// TIA Portal V17 export
FUNCTION_BLOCK "Conveyor"   // FB3, LAD
{ S7_Optimized_Access := 'TRUE' }
// Convoyeur avec démarrage temporisé
   VAR_INPUT
      Start : Bool;
      Stop : Bool;   // Arrêt (contact NF)
      Delay : Time := T#2S;
   END_VAR
   VAR_OUTPUT
      Running : Bool;
      Count : Int;
   END_VAR
   VAR
      StartTimer : TON_TIME;
      Starts : CTU_INT;
      StartEdge : Bool;
      Latched : Bool;
   END_VAR
   VAR_TEMP   // added for the SCL form of the ladder/FBD networks
      _w1 : Bool;
   END_VAR
BEGIN

REGION Network 1: Auto-maintien
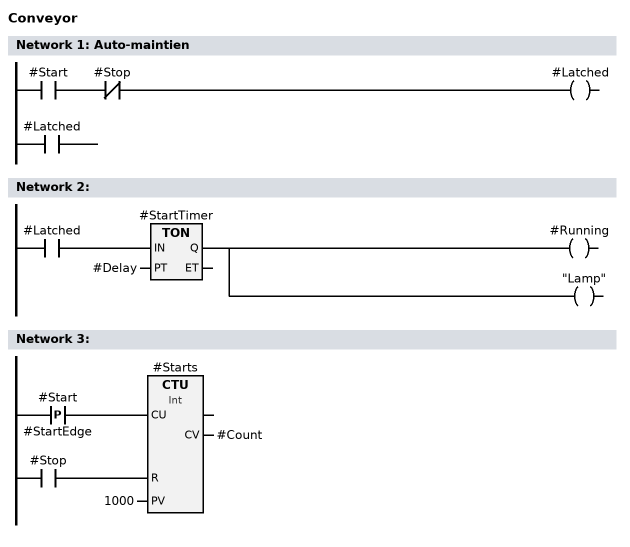
   #Latched := #Start AND NOT #Stop;
END_REGION

REGION Network 2
   RUNG wire#powerrail
      Contact( #Latched )
      #StartTimer.TON(pt := #Delay, et =>)
      wire#w1
      Coil( #Running )
   END_RUNG
   RUNG wire#w1
      Coil( "Lamp" )
   END_RUNG
   // the same network as SCL:
   #StartTimer(IN := #Latched, PT := #Delay);   // TON
   #Running := #StartTimer.Q;
   "Lamp" := #StartTimer.Q;
END_REGION

REGION Network 3
   #_w1 := #Start AND NOT #StartEdge;   // rising edge of #Start
   #StartEdge := #Start;
   #Starts(CU := #_w1, R := #Stop, PV := 1000, CV => #Count);   // CTU
END_REGION
END_FUNCTION_BLOCK
